FUNCTION_BLOCK LockingButtonWidget
VAR_INPUT
END_VAR
VAR_OUTPUT
    text : STRING;
    deactivate : BOOL;
END_VAR
VAR_IN_OUT
    status : InitializationStatus;
	lock : Process;
	unlock : Process;
END_VAR
VAR
    do_request : BOOL := FALSE;
END_VAR

IF status.locked THEN
    text := 'Unlock';
    deactivate := unlock.statuses.enabledStatus.disabled;
    
    IF do_request THEN
        unlock.request();
        do_request := FALSE;
    END_IF

ELSIF status.initialized THEN
    text := 'Lock';
    deactivate := lock.statuses.enabledStatus.disabled;
    
    IF do_request THEN
        lock.request();
        do_request := FALSE;
    END_IF
ELSE
    text := 'Unlock';
    deactivate := TRUE;
    do_request := FALSE;
END_IF

END_FUNCTION_BLOCK

(* stored: Version 1.1.0.1, ProductVersion 3.1.4018.2
   POU LockingButtonWidget: Id {2bb11438-3d3d-4851-a871-6ed6dd46ff6c}, SpecialFunc None *)
